// TwinCAT 3 PLC project IotWebSocketsSamplePostman
// ProgramVersion: 3.1.4026.11
// libraries:
//   Tc2_Standard, * (Beckhoff Automation GmbH)
//   Tc2_System, * (Beckhoff Automation GmbH)
//   Tc2_Utilities, * (Beckhoff Automation GmbH)
//   Tc3_IotBase, * (Beckhoff Automation GmbH)
// project tree:
//   DUTs/ E_State.TcDUT, FB_MyWebsocketClient.TcPOU
//   / PlcTask.TcTTO
//   POUs/ MAIN.TcPOU
// real-time tasks:
//   TASK PlcTask: cycle T#10ms, priority 20, ADS port 350

CONFIGURATION IotWebSocketsSamplePostman
    RESOURCE PLC ON TwinCAT3
        TASK PlcTask(INTERVAL := T#10ms, PRIORITY := 20);
        PROGRAM MAIN WITH PlcTask : MAIN;
    END_RESOURCE
END_CONFIGURATION

// ---- DUTs/E_State.TcDUT
{attribute 'qualified_only'}
{attribute 'strict'}
TYPE E_State :
(
	idle := 0,
	connect,
	sendMsg,
	receiveMsg,
	disconnect,
	error
) USINT;
END_TYPE

// ---- POUs/MAIN.TcPOU
PROGRAM MAIN
VAR
	eState			: E_State;
	eFailedState	: E_State;
	fbWebsocket		: FB_MyWebsocketClient;
	bConnect		: BOOL;				// set TRUE to connect and start application
	bSendMsg		: BOOL := TRUE;		// if TRUE one message will be sent
	sMessage		: STRING(255) := 'This is a message'; 	
	sMessageRcv		: STRING(255);
	nMessageRcvCnt	: UDINT;
END_VAR

CASE eState OF
E_State.idle:
	fbWebsocket.sHostName		:= 'ws.postman-echo.com';
	fbWebsocket.nHostPort		:= 443;
	fbWebsocket.sOrigin			:= 'myOrigin';
	fbWebsocket.sProtocol		:= 'myprotocol';	
	fbWebsocket.sUri			:= 'raw';
	fbWebsocket.bPerMessageDeflate := TRUE;
	fbWebsocket.stTLS.bNoServerCertCheck:=TRUE;
	
	fbWebsocket.Execute();
	IF bConnect AND NOT fbWebsocket.bConnected THEN
		eState := E_State.connect;
	END_IF
	
E_State.connect:
	IF fbWebsocket.Connect(bReconfig:=TRUE) THEN
		sMessageRcv := '';
		eState := E_State.sendMsg;
	ELSE
		eState := E_State.error;
		eFailedState := E_State.connect;
	END_IF 
	
E_State.sendMsg:
	fbWebsocket.Execute();
	IF fbWebsocket.bConnected AND bSendMsg THEN
		bSendMsg := FALSE;
		IF fbWebsocket.SendMessage(ADR(sMessage), LEN2(ADR(sMessage))+1, TRUE, TRUE) THEN 
			eState := E_State.receiveMsg; 
		ELSE
			eState := E_State.error;
			eFailedState := E_State.sendMsg;
		END_IF
	END_IF
	IF NOT bConnect THEN
		eState := E_State.disconnect;
	END_IF 
	
E_State.receiveMsg:
	fbWebsocket.Execute();
	IF NOT fbWebsocket.bConnected THEN
		eState := E_State.error;
		eFailedState := E_State.receiveMsg;
	ELSIF fbWebsocket.bMessageReceived THEN
		nMessageRcvCnt := nMessageRcvCnt+1;
		sMessageRcv := fbWebsocket.sMessage;
		bConnect := FALSE; // reset in order to disconnect (if connection should be kept open: remove this code line)
	END_IF
	IF bSendMsg THEN
		eState := E_State.sendMsg;
	END_IF
	IF NOT bConnect THEN
		eState := E_State.disconnect;
	END_IF 
	
E_State.disconnect:
	IF fbWebsocket.Disconnect() THEN
		eState := E_State.idle;
	ELSE
		eState := E_State.error;
		eFailedState := E_State.disconnect;
	END_IF

E_State.error:
	;
	
END_CASE

END_PROGRAM

// ---- DUTs/FB_MyWebsocketClient.TcPOU
{attribute 'c++_compatible'}
{attribute 'no_explicit_call' := 'do not call this POU directly'}
FUNCTION_BLOCK FB_MyWebsocketClient EXTENDS FB_IotWebSocketClient
VAR_INPUT
END_VAR
VAR_OUTPUT
	bMessageReceived	: BOOL;			// TRUE if (at least one) message was received during last execution
	sMessage			: STRING(255);	// last received message
	nMessageSize		: UDINT;		// size in bytes of last received message
	nMessageRcvCnt		: UDINT;		// count of all received messages
	nCounter:INT;
END_VAR
VAR
END_VAR

METHOD Execute
bMessageReceived := FALSE;
nMessageSize := 0;
sMessage := '';

SUPER^.Execute();
END_METHOD

{attribute 'c++_compatible'}
{attribute 'pack_mode' := '4'}
{attribute 'show'}
{attribute 'minimal_input_size' := '4'}
METHOD OnWebSocketClose : HRESULT
VAR_INPUT
	statusCode	: UINT;
	content	: PVOID;
	contentLength	: UDINT;
END_VAR
//insert business logic here

SUPER^.OnWebSocketClose(statusCode:=statusCode, content:=content, contentLength:=contentLength);
END_METHOD

{attribute 'c++_compatible'}
{attribute 'pack_mode' := '4'}
{attribute 'show'}
{attribute 'minimal_input_size' := '4'}
METHOD OnWebSocketMessage : HRESULT
VAR_INPUT
	content			: PVOID;
	contentLength	: UDINT;
	contentType		: ETcIotWebSocketContentType;
END_VAR
bMessageReceived := TRUE;
nMessageRcvCnt := nMessageRcvCnt + 1;
nMessageSize := contentLength;
IF content <> NULL AND contentLength < SIZEOF(sMessage) THEN	
	MEMSET(ADR(sMessage), 0 , SIZEOF(sMessage));	
	MEMCPY(ADR(sMessage), content, contentLength); 
END_IF

OnWebSocketMessage := SUPER^.OnWebSocketMessage(content:=content, contentLength:=contentLength, contentType:=contentType);
END_METHOD

END_FUNCTION_BLOCK
